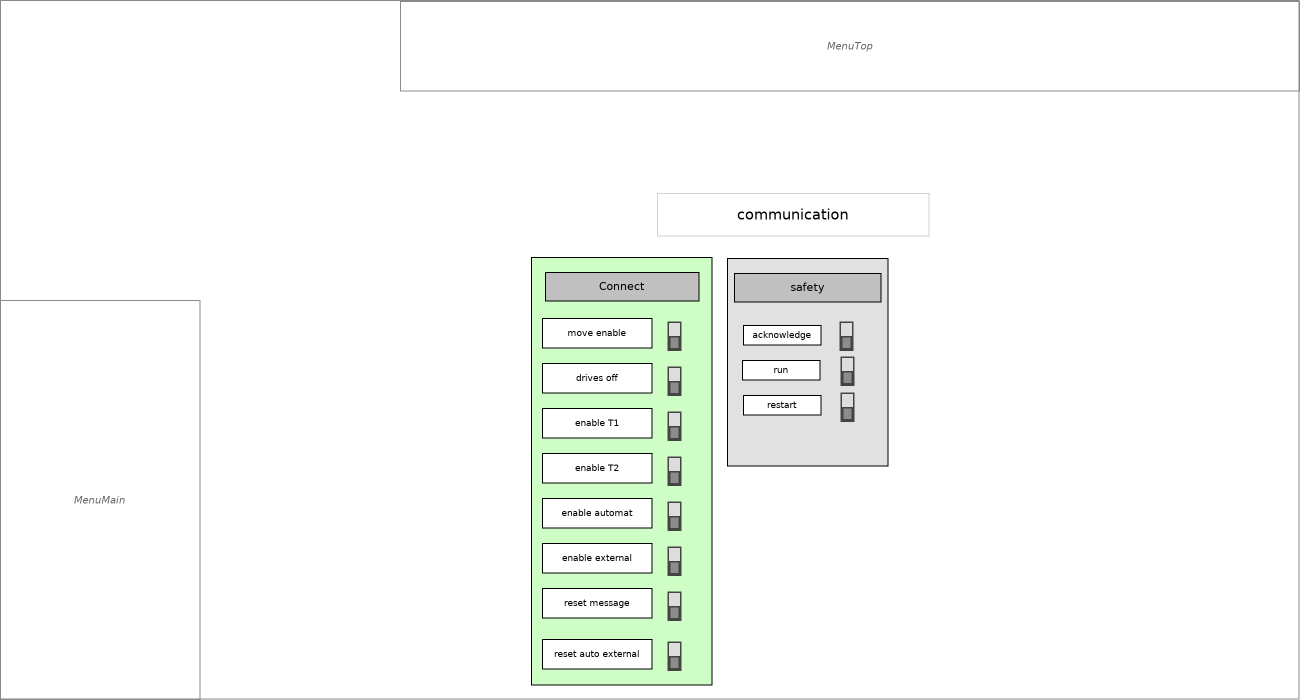
VISUALIZATION communication  // 1300x700
    Rectangle (531,257 181x428)
    Frame (400,1 900x90)
        shows MenuTop()
    Frame (0,300 200x400)
        shows MenuMain()
    Textfield (657,193 272x43), "communication"
    Rectangle (545,272 154x29), "Connect", text variable: GVL.HMI_Error_General_ID, colour toggle: GVL.HMI_Error_General
    DipSwitch (660,316 29x40), variable: MAIN.fbKRC_AutomaticExternal.MOVE_ENABLE, behaviour: TOGGLE, style: Switch-DipSwitch-Gray
    DipSwitch (660,361 29x40), variable: MAIN.fbKRC_AutomaticExternal.DRIVES_OFF, behaviour: TOGGLE, style: Switch-DipSwitch-Gray
    DipSwitch (660,406 29x40), variable: MAIN.fbKRC_AutomaticExternal.ENABLE_T1, behaviour: TOGGLE, style: Switch-DipSwitch-Gray
    DipSwitch (660,451 29x40), variable: MAIN.fbKRC_AutomaticExternal.ENABLE_T2, behaviour: TOGGLE, style: Switch-DipSwitch-Gray
    DipSwitch (660,496 29x40), variable: MAIN.fbKRC_AutomaticExternal.ENABLE_AUT, behaviour: TOGGLE, style: Switch-DipSwitch-Gray
    DipSwitch (660,541 29x40), variable: MAIN.fbKRC_AutomaticExternal.ENABLE_EXT, behaviour: TOGGLE, style: Switch-DipSwitch-Gray
    DipSwitch (660,586 29x40), variable: MAIN.fbKRC_Error.MessageReset, behaviour: TOGGLE, style: Switch-DipSwitch-Gray
    DipSwitch (660,636 29x40), variable: MAIN.fbKRC_AutomaticExternal.RESET, behaviour: TOGGLE, style: Switch-DipSwitch-Gray
    Rectangle (727,258 161x208)
    Rectangle (734,273 147x29), "safety", text variable: GVL.HMI_Error_General_ID, colour toggle: GVL.HMI_Error_General
    DipSwitch (832,316 29x40), variable: GVL_SAFETY.Ack, behaviour: TOGGLE, style: Switch-DipSwitch-Gray
    DipSwitch (833,351 29x40), variable: GVL_SAFETY.Run, behaviour: TOGGLE, style: Switch-DipSwitch-Gray
    DipSwitch (833,387 29x40), variable: GVL_SAFETY.Restart, behaviour: TOGGLE, style: Switch-DipSwitch-Gray
    Rectangle (743,325 78x20), "acknowledge"
    Rectangle (742,360 78x20), "run"
    Rectangle (743,395 78x20), "restart"
    Rectangle (542,318 110x30), "move enable"
    Rectangle (542,363 110x30), "drives off"
    Rectangle (542,408 110x30), "enable T1"
    Rectangle (542,453 110x30), "enable T2"
    Rectangle (542,498 110x30), "enable automat"
    Rectangle (542,543 110x30), "enable external"
    Rectangle (542,588 110x30), "reset message"
    Rectangle (542,639 110x30), "reset auto external"
END_VISUALIZATION

(* stored: Version 1.1.0.1, ProductVersion 3.1.4024.10
   Visu communication: Id {42cae4b6-1dcd-4029-a6b1-4c87ee3b1b78} *)
